// TIA Portal V16 export
// export: Created 2022-01-12T14:34:26.5326783Z, ExportSetting WithDefaults, DisplayName Totally Integrated Automation Portal, DisplayVersion V16 Update 4, DisplayName TIA Portal Version Control Interface, DisplayVersion V16 Update 2, DisplayName TIA Portal Openness, DisplayVersion V16 Update 4, DisplayName STEP 7 Professional, DisplayVersion V16 Update 4, DisplayName STEP 7 Safety, DisplayVersion V16, DisplayName WinCC Professional, DisplayVersion V16 Update 4
TYPE "typKlawiszeProdukcji"
// stored: IsFailsafeCompliant false
   STRUCT
      bStart { S7_SetPoint := 'True'} : "typButton";   // Aktywacja podświetla klawisz na zielono (Start pali się zawsze z innymi klawiszami)
      bPauza { S7_SetPoint := 'True'} : "typButton";   // Przytrzymanie Klawisza aktywuje K6700 (program musi pamiętać z jakiego kroku wyszedł/do jakiego ma wrócić)
      bStop { S7_SetPoint := 'True'} : "typButton";   // Przytrzymanie przez 5s K6100
      bProdukcja { S7_SetPoint := 'True'} : "typButton";   // aktywacja podświetla klawisz na zielono
      bCyrkulacja { S7_SetPoint := 'True'} : "typButton";   // aktywacja podświetla klawisz na żółto; awaryjnie na czerwono
      bCip { S7_SetPoint := 'True'} : "typButton";   // aktywacja podświetla klawisz na zielono
      bPullout { S7_SetPoint := 'True'} : "typButton";   // aktywacja podświetla klawisz na zielono
      bFlux { S7_SetPoint := 'True'} : "typButton";
      bNastepnyKrok { S7_SetPoint := 'True'} : "typButton";   // nastepny krok wyskakuje podczas mycia jezeli alarm 18
      bPrzygotowanie { S7_SetPoint := 'True'} : "typButton";   // przygotowanie stacji CIP
   END_STRUCT;
END_TYPE
